% RSLogix 500 project P5_ROTOMETER.RSS, saved by version 8.30.00.16 %
PROJECT "P5"    % processor: Bul.1763 MicroLogix 1100 Series B %

PROGRAM FILES
  LAD 2   6 rungs

DATA FILES
  O0 OUTPUT  4 elements
  I1 INPUT  6 elements
  S2 STATUS  66 elements
  B3 BINARY  1 elements
  T4 TIMER  3 elements
  C5 COUNTER  1 elements
  R6 CONTROL  1 elements
  N7 INTEGER  1 elements
  F8 FLOAT  3 elements

LADDER 2
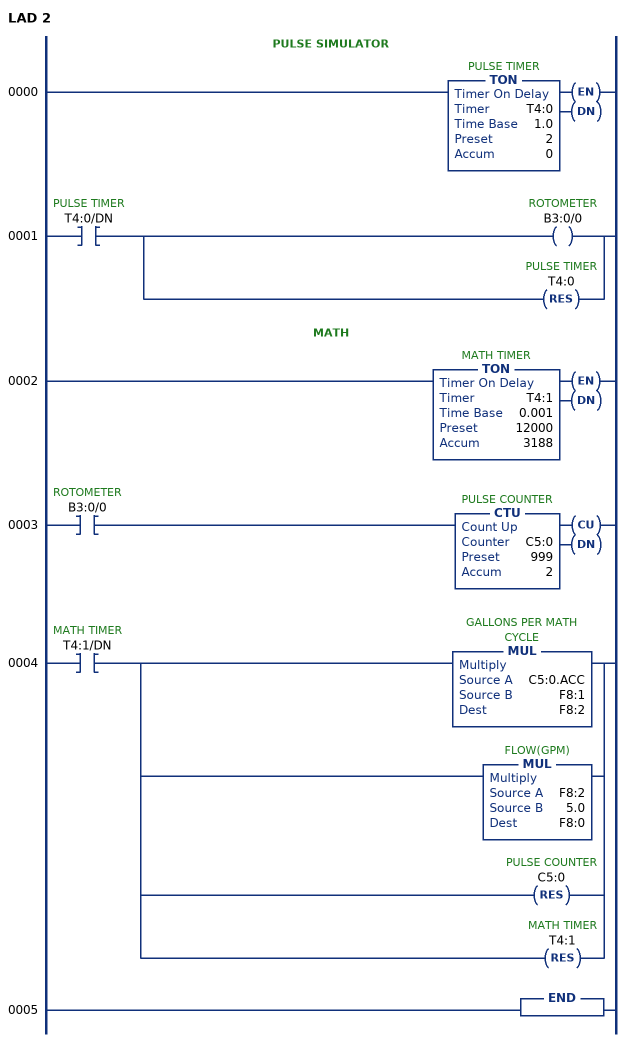
% Rung: 0 %
% TITLE: PULSE SIMULATOR %
SOR TON T4:0 1.0 2 0 EOR
%   T4:0  "PULSE TIMER" %
% Rung: 1 %
SOR XIC T4:0/DN BST OTE B3:0/0 NXB RES T4:0 BND EOR
%   T4:0  "PULSE TIMER" %
%   B3:0/0  "ROTOMETER" %
% Rung: 2 %
% TITLE: MATH %
SOR TON T4:1 0.001 12000 3188 EOR
%   T4:1  "MATH TIMER" %
% Rung: 3 %
SOR XIC B3:0/0 CTU C5:0 999 2 EOR
%   B3:0/0  "ROTOMETER" %
%   C5:0  "PULSE COUNTER" %
% Rung: 4 %
SOR XIC T4:1/DN BST MUL C5:0.ACC F8:1 F8:2 NXB MUL F8:2 5.0 F8:0 NXB RES C5:0 NXB RES T4:1 BND EOR
%   T4:1  "MATH TIMER" %
%   C5:0  "PULSE COUNTER" %
%   F8:1  "FLOW (GPP)" %
%   F8:2  "GALLONS PER MATH CYCLE" %
%   F8:0  "FLOW(GPM)" %
% Rung: 5 %
SOR END EOR

OTHER DOCUMENTED ADDRESSES
  N7:0  "PPM"

DATA TABLE (non-zero values as saved)
DATA T4
% .PRE .ACC %
% T4:0 % 2 0
% T4:1 % 12000 3188
DATA C5
% .PRE .ACC %
% C5:0 % 999 2
DATA F8
% F8:0 % 189 6.3 37.8
